# EPICS alarm handler configuration: mps_database/bareTest/alarms/areas/mpln_bpn15_mp01.alhConfig
GROUP NULL MPLN:BPN15:MP01:1
$ALIAS MPS Link Node 79
$GUIDANCE
LTUH MPS
   Group Name: MPLN:BPN15:MP01:1
   Summary PV:  MPLN:BPN15:MP01:1:STATSUMY
$END
CHANNEL  MPLN:BPN15:MP01:1    MPLN:BPN15:MP01:1:MPS_EN_RBV		-----
CHANNEL  MPLN:BPN15:MP01:1    MPLN:BPN15:MP01:1:LC1_MODE_RBV		-----
